// Manages symbols paths, supporting segment-based navigation, validation, and modification.
// Example path: MAIN.functionBlock.5.bBool
FUNCTION_BLOCK FINAL TagPath
VAR
	_sPath		: Str;
	_nLen		: INT := 0;
	_nSegStart	: INT := 0;
	_nSegEnd	: INT := 0;
END_VAR

METHOD PRIVATE _HasIncorrectSymbols : BOOL
VAR_INPUT
	sToCheck		: Str;
END_VAR
VAR
	i				: INT;
	_nStrLen		: INT := Tc2_Standard.LEN(sToCheck);
	_sChar			: Ch;
END_VAR
_sChar := Tc2_Standard.MID(sToCheck, 1, 1);
IF (_sChar >= '0') AND (_sChar <= '9') THEN
    _HasIncorrectSymbols := TRUE; // Cannot start with a number
    RETURN;
END_IF;

// Loop through the rest of the string to validate each character
FOR i := 1 TO _nStrLen DO
    _sChar := Tc2_Utilities.F_ToLCase(Tc2_Standard.MID(sToCheck, 1, i));
    
    // Check for invalid characters
    IF NOT ((_sChar >= 'a' AND _sChar <= 'z') OR 	// Lowercase letters
            (_sChar >= '0' AND _sChar <= '9') OR 	// Numbers
            (_sChar = '_') OR                 		// Underscore
			(_sChar = '*')) THEN					// Wildcard
        _HasIncorrectSymbols := TRUE; // Invalid character found
        RETURN;
    END_IF;
END_FOR;

// If no invalid characters are found, return FALSE
_HasIncorrectSymbols := FALSE;
END_METHOD

// Adds a new segment to the path after the current segment.
// Returns `Ok` if successful, `None` if invalid.
METHOD AddNext : Result
VAR_INPUT
    sToAdd : Str; // Segment to add
END_VAR
VAR
	_nNewLen	: INT := _nLen + Tc2_Standard.LEN(sToAdd) + 1;
END_VAR
IF _sPath = '' OR _nSegStart = 0 OR sToAdd = '' THEN
    AddNext := None;
    RETURN;
END_IF;

IF _HasIncorrectSymbols(sToAdd) THEN
	AddNext := None;
	RETURN;
END_IF

IF _nNewLen <= 255 THEN
	_sPath := Tc2_Standard.INSERT(_sPath, '.', _nSegEnd);
	_sPath := Tc2_Standard.INSERT(_sPath, sToAdd, _nSegEnd + 1);
	_nLen := _nNewLen;
	AddNext := Ok;
END_IF
END_METHOD

// Adds a new segment to the path before the current segment.
// Returns `Ok` if successful, `None` if invalid.
METHOD AddPrev : Result
VAR_INPUT
    sToAdd : Str; // Segment to add
END_VAR
VAR
	_nAddLen	: INT := Tc2_Standard.LEN(sToAdd);
	_nNewLen	: INT := _nLen + _nAddLen + 1;
END_VAR
IF _sPath = '' OR _nSegStart = 0 OR sToAdd = '' THEN
    AddPrev := None;
    RETURN;
END_IF;

IF _HasIncorrectSymbols(sToAdd) THEN
	AddPrev := None;
	RETURN;
END_IF

IF _nNewLen <= 255 THEN
	_sPath := Tc2_Standard.INSERT(_sPath, '.', _nSegStart - 1);
	_sPath := Tc2_Standard.INSERT(_sPath, sToAdd, _nSegStart - 2);
	_nLen := _nNewLen;
	_nSegStart := _nSegStart + _nAddLen + 1;
	_nSegEnd := _nSegEnd + _nAddLen + 1;
	AddPrev := Ok;
END_IF
END_METHOD

// Retrieves the current segment from the path.
// Returns `Ok` if successful, `None` if no segment is found.
METHOD Get : Result
VAR_OUTPUT
    sSeg : Str; // Current segment
END_VAR
IF _nSegStart = 0 THEN
	RETURN;
END_IF

sSeg := Tc2_Standard.MID(_sPath, _nSegEnd - _nSegStart + 1, _nSegStart);
IF sSeg <> '' THEN
	Get := Ok;
END_IF
END_METHOD

// Moves to the next segment in the path and retrieves it.
// Returns `Ok` if successful, `None` if no next segment exists.
METHOD Next : Result
VAR_OUTPUT
    sSeg : Str; // Next segment
END_VAR
VAR
	i			: INT;
END_VAR
// If the path is invalid or already fully processed
IF _sPath = '' OR _nSegEnd = _nLen THEN
    Next := None;
    RETURN;
END_IF;

// Initialize on the first call
IF _nSegStart = 0 THEN
    _nSegStart := 1;
    FOR i := 1 TO _nLen DO
        IF Tc2_Standard.MID(_sPath, 1, i) = '.' THEN
            _nSegEnd := i - 1;
            EXIT;
        END_IF;
    END_FOR;

	IF _nSegEnd < _nSegStart THEN
		_nSegEnd := _nLen;
	END_IF;

    sSeg := Tc2_Standard.MID(_sPath, _nSegEnd - _nSegStart + 1, _nSegStart);
    Next := Ok;
    RETURN;
END_IF;

_nSegStart := _nSegEnd + 2; // Skip the delimiter

FOR i := _nSegStart TO _nLen DO
    IF Tc2_Standard.MID(_sPath, 1, i) = '.' THEN
        _nSegEnd := i - 1;
        EXIT;
    END_IF;
END_FOR;

// If no more delimiters, this is the last segment
IF _nSegEnd < _nSegStart THEN
    _nSegEnd := _nLen;
END_IF;

sSeg := Tc2_Standard.MID(_sPath, _nSegEnd - _nSegStart + 1, _nSegStart);
Next := Ok;
END_METHOD

// Retrieves the next segment without moving the segment pointer.
// Returns Ok if successful, None if no next segment exists.
METHOD Peek : Result
VAR_OUTPUT
    sSeg : Str; // Next segment
END_VAR
VAR
	i			: INT;
	_nPeekStart	: INT := 0;
	_nPeekEnd	: INT := 0;
END_VAR
// If the path is invalid or already fully processed
IF _sPath = '' OR _nSegEnd = _nLen OR _nSegStart = 0 THEN
    Peek := None;
    RETURN;
END_IF;

_nPeekStart := _nSegEnd + 2; // Skip the delimiter

FOR i := _nPeekStart TO _nLen DO
    IF Tc2_Standard.MID(_sPath, 1, i) = '.' THEN
        _nPeekEnd := i - 1;
        EXIT;
    END_IF;
END_FOR;

// If no more delimiters, this is the last segment
IF _nPeekEnd = 0 THEN
    _nPeekEnd := _nLen;
END_IF;

sSeg := Tc2_Standard.MID(_sPath, _nPeekEnd - _nPeekStart + 1, _nPeekStart);
Peek := Ok;
END_METHOD

// Retrieves the previous segment without moving the segment pointer.
// Returns `Ok` if successful, `None` if no previous segment exists.
METHOD PeekBack : Result
VAR_OUTPUT
    sSeg : Str; // Previous segment
END_VAR
VAR
	i			: INT;
	_nPeekStart	: INT := 0;
	_nPeekEnd	: INT := 0;
END_VAR
// If the path is invalid or already fully processed
IF _sPath = '' OR _nSegEnd = 0 OR _nSegStart = 1 THEN
    PeekBack := None;
    RETURN;
END_IF;

_nPeekEnd := _nSegStart - 2; // Skip the delimiter

FOR i := _nPeekEnd TO 1 BY -1 DO
    IF Tc2_Standard.MID(_sPath, 1, i) = '.' THEN
        _nPeekStart := i + 1;
        EXIT;
    END_IF;
END_FOR;

// If no more delimiters, this is the first segment
IF _nPeekStart = 0 THEN
    _nPeekStart := 1;
END_IF;

sSeg := Tc2_Standard.MID(_sPath, _nPeekEnd - _nPeekStart + 1, _nPeekStart);
PeekBack := Ok;
END_METHOD

// Moves to the previous segment in the path and retrieves it.
// Returns `Ok` if successful, `None` if no previous segment exists.
METHOD Prev : Result
VAR_OUTPUT
    sSeg : Str; // Previous segment
END_VAR
VAR
	i			: INT;
END_VAR
// If the path is invalid or already fully processed
IF _sPath = '' OR _nSegStart = 1 THEN
    Prev := None;
    RETURN;
END_IF;

// Initialize on the first call
IF _nSegEnd = 0 THEN
    _nSegEnd := _nLen;
    FOR i := _nSegEnd TO 1 BY -1 DO
        IF Tc2_Standard.MID(_sPath, 1, i) = '.' THEN
            _nSegStart := i + 1;
            EXIT;
        END_IF;
    END_FOR;

	// If no more delimiters, this is the first segment
	IF _nSegEnd < _nSegStart THEN
		_nSegStart := 1;
	END_IF;

    sSeg := Tc2_Standard.MID(_sPath, _nSegEnd - _nSegStart + 1, _nSegStart);
    Prev := Ok;
    RETURN;
END_IF;

_nSegEnd := _nSegStart - 2; // Skip the delimiter

FOR i := _nSegEnd TO 1 BY -1 DO
    IF Tc2_Standard.MID(_sPath, 1, i) = '.' THEN
        _nSegStart := i + 1;
        EXIT;
    END_IF;
END_FOR;

// If no more delimiters, this is the first segment
IF _nSegEnd < _nSegStart THEN
    _nSegStart := 1;
END_IF;

sSeg := Tc2_Standard.MID(_sPath, _nSegEnd - _nSegStart + 1, _nSegStart);
Prev := Ok;
END_METHOD

// Reads and returns the entire symbolic path as a string.
METHOD Read : Str
Read := _sPath;
END_METHOD

// Removes the current segment and moves to the next segment.
// Returns `Ok` if successful, `None` if no segment to remove.
METHOD RemoveAndNext : Result
VAR
    _nSegLen		: INT := _nSegEnd - _nSegStart + 1; // Length of the segment to remove
    _bIsFirstSeg	: BOOL := (_nSegStart = 1); // Check if the segment is the first segment
    _bIsLastSeg		: BOOL := (_nSegEnd = _nLen); // Check if the segment is the last segment
	i				: INT;
END_VAR
// Ensure the current path is valid
IF _sPath = '' OR _nSegStart = 0 THEN
    RemoveAndNext := None;
    RETURN;
END_IF;

IF _bIsFirstSeg AND _bIsLastSeg THEN	
	_sPath := '';
    _nLen := 0;
	_nSegStart := 0;
	_nSegEnd := 0;
	RemoveAndNext := Ok;
ELSIF _bIsFirstSeg THEN
	_sPath := Tc2_Standard.DELETE(_sPath, _nSegLen + 1, _nSegStart); // Also removes dot after first segment
	_nLen := _nLen - _nSegLen;
	_nSegStart := 0;
	_nSegEnd := 0;
	RemoveAndNext := Ok;
ELSIF _bIsLastSeg THEN
	_sPath := Tc2_Standard.DELETE(_sPath, _nSegLen + 1, _nSegStart - 1); // Also removes dot before last segment
	_nLen := _nLen - _nSegLen;
	_nSegStart := 0;
	_nSegEnd := 0;
	RemoveAndNext := Ok;
ELSE
	_sPath := Tc2_Standard.DELETE(_sPath, _nSegLen + 1, _nSegStart); // Also removes dot after segment
	_nLen := _nLen - _nSegLen;
	_nSegStart := _nSegEnd + 2; // Skip the delimiter
	
	FOR i := _nSegStart TO _nLen DO
		IF Tc2_Standard.MID(_sPath, 1, i) = '.' THEN
			_nSegEnd := i - 1;
			EXIT;
		END_IF;
	END_FOR;
	
	// If no more delimiters, this is the last segment
	IF _nSegEnd < _nSegStart THEN
		_nSegEnd := _nLen;
	END_IF;
	RemoveAndNext := Ok;
END_IF
END_METHOD

// Removes the current segment and moves to the previous segment.
// Returns `Ok` if successful, `None` if no segment to remove.
METHOD RemoveAndPrev : Result
VAR
    _nSegLen		: INT := _nSegEnd - _nSegStart + 1; // Length of the segment to remove
    _bIsFirstSeg	: BOOL := (_nSegStart = 1); // Check if the segment is the first segment
    _bIsLastSeg		: BOOL := (_nSegEnd = _nLen); // Check if the segment is the last segment
	i				: INT;
END_VAR
// Ensure the current path is valid
IF _sPath = '' OR _nSegStart = 0 THEN
    RemoveAndPrev := None;
    RETURN;
END_IF;

IF _bIsFirstSeg AND _bIsLastSeg THEN	
	_sPath := '';
    _nLen := 0;
	_nSegStart := 0;
	_nSegEnd := 0;
	RemoveAndPrev := Ok;
ELSIF _bIsFirstSeg THEN
	_sPath := Tc2_Standard.DELETE(_sPath, _nSegLen + 1, _nSegStart); // Also removes dot after first segment
	_nLen := _nLen - _nSegLen;
	_nSegStart := 0;
	_nSegEnd := 0;
	RemoveAndPrev := Ok;
ELSIF _bIsLastSeg THEN
	_sPath := Tc2_Standard.DELETE(_sPath, _nSegLen + 1, _nSegStart - 1); // Also removes dot before last segment
	_nLen := _nLen - _nSegLen;
	_nSegStart := 0;
	_nSegEnd := 0;
	RemoveAndPrev := Ok;
ELSE
	_sPath := Tc2_Standard.DELETE(_sPath, _nSegLen + 1, _nSegStart); // Also removes dot after segment
	_nLen := _nLen - _nSegLen;
	_nSegEnd := _nSegStart - 2; // Skip the delimiter
	
	FOR i := _nSegEnd TO 1 BY -1 DO
		IF Tc2_Standard.MID(_sPath, 1, i) = '.' THEN
			_nSegStart := i + 1;
			EXIT;
		END_IF;
	END_FOR;
	
	// If no more delimiters, this is the first segment
	IF _nSegEnd < _nSegStart THEN
		_nSegStart := 1;
	END_IF;
	RemoveAndPrev := Ok;
END_IF
END_METHOD

// Sets the symbolic path to a new value.
// Validates the input path for correctness.
// Returns `Ok` if successful, `None` if invalid.
METHOD Set : Result
VAR_INPUT
    sNewPath : Str; // New path to set
END_VAR

VAR
	i				: INT;
	_nStrLen		: INT := Tc2_Standard.LEN(sNewPath);
	_sChar			: Ch;
END_VAR
IF sNewPath = '' THEN
	Set := None;
	RETURN;
END_IF

_sChar := Tc2_Standard.MID(sNewPath, 1, 1);
IF (_sChar >= '0') AND (_sChar <= '9') THEN
	Set := None;
    RETURN;
END_IF;

sNewPath := Tc2_Utilities.F_ToLCase(sNewPath);

FOR i := 1 TO _nStrLen DO
    _sChar := Tc2_Standard.MID(sNewPath, 1, i);
    
    // Check for invalid characters
    IF NOT ((_sChar >= 'a' AND _sChar <= 'z') OR 	// Lowercase letters
            (_sChar >= '0' AND _sChar <= '9') OR 	// Numbers
            (_sChar = '_') OR                 		// Underscore
			(_sChar = '.') OR
			(_sChar = '*')) THEN					// Wildcard
		Set := None;
        RETURN;
    END_IF;
END_FOR;

IF Tc2_Standard.FIND(sNewPath, '..') <> 0 THEN
	Set := None;
	RETURN;
END_IF

IF Tc2_Standard.FIND(sNewPath, '**') <> 0 THEN
	Set := None;
	RETURN;
END_IF

_sPath := sNewPath;
_nLen := _nStrLen;
Set := Ok;
END_METHOD

// Replaces the current segment with a new segment.
// Returns `Ok` if successful, `None` if invalid.
METHOD Swap : Result
VAR_INPUT
    sToSwap : Str; // New segment to replace the current segment
END_VAR
VAR
	_nSegLen	: INT := _nSegEnd - _nSegStart + 1;
	_nSwapLen	: INT := Tc2_Standard.LEN(sToSwap);
	_nNewLen	: INT := _nLen - _nSegLen + _nSwapLen;
END_VAR
IF _sPath = '' OR _nSegStart = 0 OR sToSwap = '' THEN
    Swap := None;
    RETURN;
END_IF;

IF _HasIncorrectSymbols(sToSwap) THEN
	Swap := None;
	RETURN;
END_IF

IF _nNewLen <= 255 THEN
	_sPath := Tc2_Standard.REPLACE(_sPath, sToSwap, _nSegLen, _nSegStart);
	_nSegEnd := _nSegStart + _nSwapLen - 1;
	_nLen := _nNewLen;
	Swap := Ok;
END_IF
END_METHOD

END_FUNCTION_BLOCK

(* stored: Version 1.1.0.1
   POU TagPath: Id {de08c266-82f2-43b6-8ef2-f01293adb92c}, SpecialFunc None
   Method _HasIncorrectSymbols: Id {7921e82a-db38-44ae-a783-6bcceb0d9a9c}
   Method AddNext: Id {5c98e624-d0b2-49a6-83ae-ef070e544a65}
   Method AddPrev: Id {f37fed9e-731e-4322-bff5-14304a710b2b}
   Method Get: Id {3e3a2b44-c68d-43c1-ba42-e4a27a76ea9b}
   Method Next: Id {c6cdf833-e7f8-4994-a776-e72dded77005}
   Method Peek: Id {644fd812-0eb6-44b1-9b5a-072d8067b266}
   Method PeekBack: Id {f7303771-b30b-4296-89fd-270bf803a6c6}
   Method Prev: Id {bb912db9-78e6-4226-9a9c-08a0cddabbba}
   Method Read: Id {178f264a-e89a-4d3a-b8d2-3ca5f74b3ae7}
   Method RemoveAndNext: Id {0d255a40-6614-4f67-94dc-6238407c06a7}
   Method RemoveAndPrev: Id {c1a28866-c26a-4715-bc3f-11af169f2834}
   Method Set: Id {59eb7151-fecf-4492-8bf1-30025d8074fd}
   Method Swap: Id {cc9e4235-2aed-4cdd-a813-c026de498a1d} *)
